INTERFACE ITF_TaskAllocation

METHOD Invoke
VAR_INPUT
END_VAR
END_METHOD

PROPERTY Task : E_Task
GET
END_GET
SET
END_SET
END_PROPERTY

PROPERTY TaskId : Int
GET
END_GET
SET
END_SET
END_PROPERTY

END_INTERFACE

(* stored: Version 1.1.0.1, ProductVersion 3.1.4022.7
   Itf ITF_TaskAllocation: Id {68b780d1-bd30-481c-b84c-a2476551ddbd}
   Method Invoke: Id {d1e24f08-e42d-4606-87bd-13c61275799a}
   Property Task: Id {1abf0074-5672-460a-898b-904f839e1bb5}
   Get Get: Id {a7086290-0635-4e73-8ee4-a51b8d25bc93}
   Set Set: Id {cad807d8-0700-4768-9055-77ae9f35ec82}
   Property TaskId: Id {0ccf2a85-ca5a-440e-b527-3ac6027bb270}
   Get Get: Id {fa83aced-722a-4d9f-a630-32b235f2685c}
   Set Set: Id {601e229b-8097-4be9-85b9-4fed0194d03b} *)
